// TIA Portal project "Bol1" (V17)

(* hardware
DEVICE "S7-1200 station_1"  S7-1200 Station
   slot 0: "Rack_0"  S7-1200 Rack  Rack  V1.0
   slot 1: "PLC_1"  CPU 1214C AC/DC/Rly  6ES7 214-1BG40-0XB0  V4.5
*)

// ===== PLC "PLC_1"  CPU 1214C AC/DC/Rly =====

VAR_GLOBAL   // PLC tag table "Tabla de variables estándar"
   "Ent0" AT %I0.0 : Bool;
   "Ent1" AT %I0.1 : Bool;
   "Ent2" AT %I0.2 : Bool;
   "Ent3" AT %I0.3 : Bool;
   "Out0" AT %Q0.0 : Bool;
   "Out1" AT %Q0.1 : Bool;
   "Out2" AT %Q0.2 : Bool;
   "Out3" AT %Q0.3 : Bool;
   "Ent4" AT %I0.4 : Bool;
   "Out4" AT %Q0.4 : Bool;
   "Tag_1" AT %M2.2 : Bool;
END_VAR

DATA_BLOCK "Bloque"   // DB1
{ S7_Optimized_Access := 'TRUE' }
VERSION : 0.1
   VAR
      A0 : Array[0..4] of Bool;
      A1 : Array[0..4] of Bool;
      A2 : Array[0..4] of Bool;
      A3 : Array[0..4] of Bool;
      A4 : Array[0..4] of Bool;
      S : Array[0..4] of Bool;
   END_VAR
BEGIN
END_DATA_BLOCK

ORGANIZATION_BLOCK "Main"   // OB1, LAD, ProgramCycle
TITLE = "Main Program Sweep (Cycle)"
{ S7_Optimized_Access := 'TRUE' }
VERSION : 0.1
   VAR_INPUT
      Initial_Call : Bool;   // Initial call of this OB
      Remanence : Bool;   // =True, if remanent data are available
   END_VAR
BEGIN

REGION Network 1
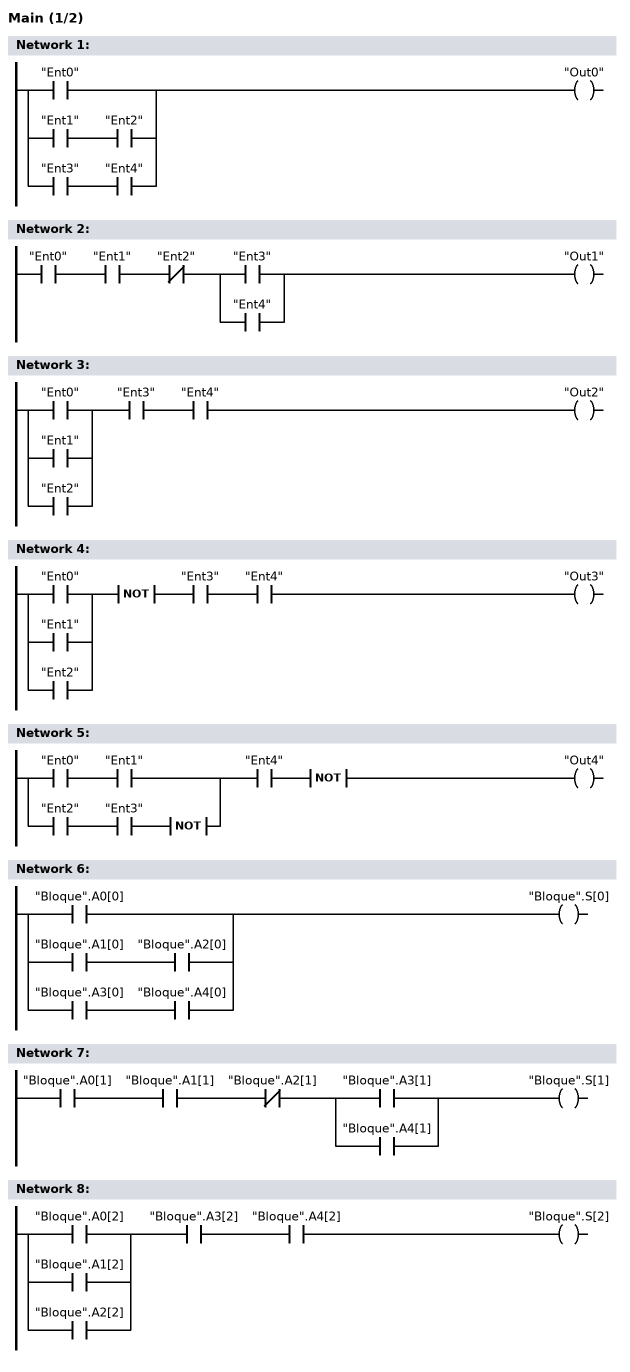
   RUNG wire#powerrail
      Contact( "Ent0" )
      wire#w1
      Coil( "Out0" )
   END_RUNG
   RUNG wire#powerrail
      Contact( "Ent1" )
      Contact( "Ent2" )
   END_RUNG wire#w1
   RUNG wire#powerrail
      Contact( "Ent3" )
      Contact( "Ent4" )
   END_RUNG wire#w1
   // the same network as SCL:
   "Out0" := "Ent0" OR ("Ent1" AND "Ent2") OR ("Ent3" AND "Ent4");
END_REGION

REGION Network 2
   RUNG wire#powerrail
      Contact( "Ent0" )
      Contact( "Ent1" )
      I_Contact( "Ent2" )
      wire#w1
      Contact( "Ent3" )
      wire#w2
      Coil( "Out1" )
   END_RUNG
   RUNG wire#w1
      Contact( "Ent4" )
   END_RUNG wire#w2
   // the same network as SCL:
   "Out1" := "Ent0" AND "Ent1" AND NOT "Ent2" AND ("Ent3" OR "Ent4");
END_REGION

REGION Network 3
   RUNG wire#powerrail
      Contact( "Ent0" )
      wire#w1
      Contact( "Ent3" )
      Contact( "Ent4" )
      Coil( "Out2" )
   END_RUNG
   RUNG wire#powerrail
      Contact( "Ent1" )
   END_RUNG wire#w1
   RUNG wire#powerrail
      Contact( "Ent2" )
   END_RUNG wire#w1
   // the same network as SCL:
   "Out2" := ("Ent0" OR "Ent1" OR "Ent2") AND "Ent3" AND "Ent4";
END_REGION

REGION Network 4
   RUNG wire#powerrail
      Contact( "Ent0" )
      wire#w1
      Not()
      Contact( "Ent3" )
      Contact( "Ent4" )
      Coil( "Out3" )
   END_RUNG
   RUNG wire#powerrail
      Contact( "Ent1" )
   END_RUNG wire#w1
   RUNG wire#powerrail
      Contact( "Ent2" )
   END_RUNG wire#w1
   // the same network as SCL:
   "Out3" := NOT ("Ent0" OR "Ent1" OR "Ent2") AND "Ent3" AND "Ent4";
END_REGION

REGION Network 5
   RUNG wire#powerrail
      Contact( "Ent0" )
      Contact( "Ent1" )
      wire#w1
      Contact( "Ent4" )
      Not()
      Coil( "Out4" )
   END_RUNG
   RUNG wire#powerrail
      Contact( "Ent2" )
      Contact( "Ent3" )
      Not()
   END_RUNG wire#w1
   // the same network as SCL:
   "Out4" := NOT ((("Ent0" AND "Ent1") OR NOT ("Ent2" AND "Ent3")) AND "Ent4");
END_REGION

REGION Network 6
   RUNG wire#powerrail
      Contact( "Bloque".A0[0] )
      wire#w1
      Coil( "Bloque".S[0] )
   END_RUNG
   RUNG wire#powerrail
      Contact( "Bloque".A1[0] )
      Contact( "Bloque".A2[0] )
   END_RUNG wire#w1
   RUNG wire#powerrail
      Contact( "Bloque".A3[0] )
      Contact( "Bloque".A4[0] )
   END_RUNG wire#w1
   // the same network as SCL:
   "Bloque".S[0] := "Bloque".A0[0] OR ("Bloque".A1[0] AND "Bloque".A2[0]) OR ("Bloque".A3[0] AND "Bloque".A4[0]);
END_REGION

REGION Network 7
   RUNG wire#powerrail
      Contact( "Bloque".A0[1] )
      Contact( "Bloque".A1[1] )
      I_Contact( "Bloque".A2[1] )
      wire#w1
      Contact( "Bloque".A3[1] )
      wire#w2
      Coil( "Bloque".S[1] )
   END_RUNG
   RUNG wire#w1
      Contact( "Bloque".A4[1] )
   END_RUNG wire#w2
   // the same network as SCL:
   "Bloque".S[1] := "Bloque".A0[1] AND "Bloque".A1[1] AND NOT "Bloque".A2[1] AND ("Bloque".A3[1] OR "Bloque".A4[1]);
END_REGION

REGION Network 8
   RUNG wire#powerrail
      Contact( "Bloque".A0[2] )
      wire#w1
      Contact( "Bloque".A3[2] )
      Contact( "Bloque".A4[2] )
      Coil( "Bloque".S[2] )
   END_RUNG
   RUNG wire#powerrail
      Contact( "Bloque".A1[2] )
   END_RUNG wire#w1
   RUNG wire#powerrail
      Contact( "Bloque".A2[2] )
   END_RUNG wire#w1
   // the same network as SCL:
   "Bloque".S[2] := ("Bloque".A0[2] OR "Bloque".A1[2] OR "Bloque".A2[2]) AND "Bloque".A3[2] AND "Bloque".A4[2];
END_REGION

REGION Network 9
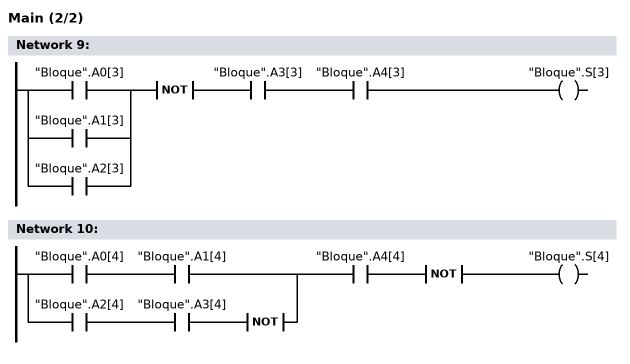
   RUNG wire#powerrail
      Contact( "Bloque".A0[3] )
      wire#w1
      Not()
      Contact( "Bloque".A3[3] )
      Contact( "Bloque".A4[3] )
      Coil( "Bloque".S[3] )
   END_RUNG
   RUNG wire#powerrail
      Contact( "Bloque".A1[3] )
   END_RUNG wire#w1
   RUNG wire#powerrail
      Contact( "Bloque".A2[3] )
   END_RUNG wire#w1
   // the same network as SCL:
   "Bloque".S[3] := NOT ("Bloque".A0[3] OR "Bloque".A1[3] OR "Bloque".A2[3]) AND "Bloque".A3[3] AND "Bloque".A4[3];
END_REGION

REGION Network 10
   RUNG wire#powerrail
      Contact( "Bloque".A0[4] )
      Contact( "Bloque".A1[4] )
      wire#w1
      Contact( "Bloque".A4[4] )
      Not()
      Coil( "Bloque".S[4] )
   END_RUNG
   RUNG wire#powerrail
      Contact( "Bloque".A2[4] )
      Contact( "Bloque".A3[4] )
      Not()
   END_RUNG wire#w1
   // the same network as SCL:
   "Bloque".S[4] := NOT ((("Bloque".A0[4] AND "Bloque".A1[4]) OR NOT ("Bloque".A2[4] AND "Bloque".A3[4])) AND "Bloque".A4[4]);
END_REGION
END_ORGANIZATION_BLOCK